Omron CX-Programmer project NewProject (CX-Programmer 9.81)

# PLC NewPLC1: CJ2M CPU11

## Program NewProgram1 (cyclic task 0)
Local symbols
Int_1 0.00 BOOL  ; Interruptor 1
Int_2 0.01 BOOL  ; Interruptor 2
Lampada_1 1.00 BOOL  ; Lampada 1
Lampada_2 1.01 BOOL  ; Lampada 2
Lampada_3 1.02 BOOL  ; Lampada 3
Lampada_4 1.03 BOOL  ; Lampada 4

### Section Section1

### Section Outputs

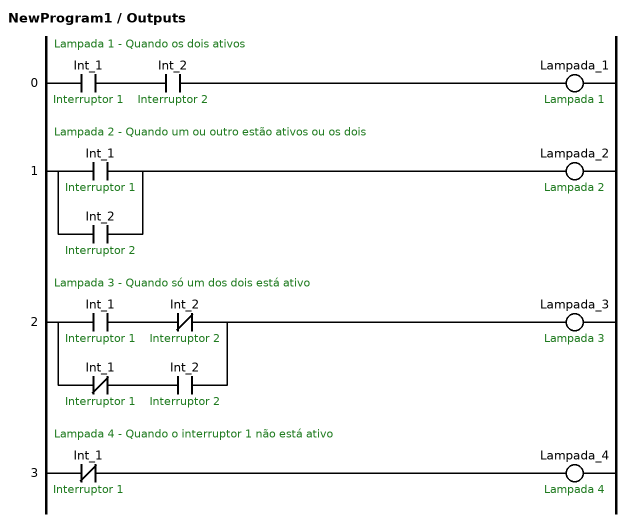
; rung 0: Lampada 1 - Quando os dois ativos
LD Int_1  ; Interruptor 1
AND Int_2  ; Interruptor 2
OUT Lampada_1  ; Lampada 1
; rung 1: Lampada 2 - Quando um ou outro estão ativos ou os dois
LD Int_1  ; Interruptor 1
OR Int_2  ; Interruptor 2
OUT Lampada_2  ; Lampada 2
; rung 2: Lampada 3 - Quando só um dos dois está ativo
LD Int_1  ; Interruptor 1
ANDNOT Int_2  ; Interruptor 2
LDNOT Int_1  ; Interruptor 1
AND Int_2  ; Interruptor 2
ORLD
OUT Lampada_3  ; Lampada 3
; rung 3: Lampada 4 - Quando o interruptor 1 não está ativo
LDNOT Int_1  ; Interruptor 1
OUT Lampada_4  ; Lampada 4

### Section END
; rung 0
END(001)